// TIA Portal V19 export
FUNCTION "RO_2" : Void   // FC11, LAD
{ S7_Optimized_Access := 'TRUE' }
// stored: SetENOAutomatically false
   VAR_TEMP   // added for the SCL form of the ladder/FBD networks
      _w1 : Bool;
   END_VAR
BEGIN

REGION Network 1: FEED PUMP
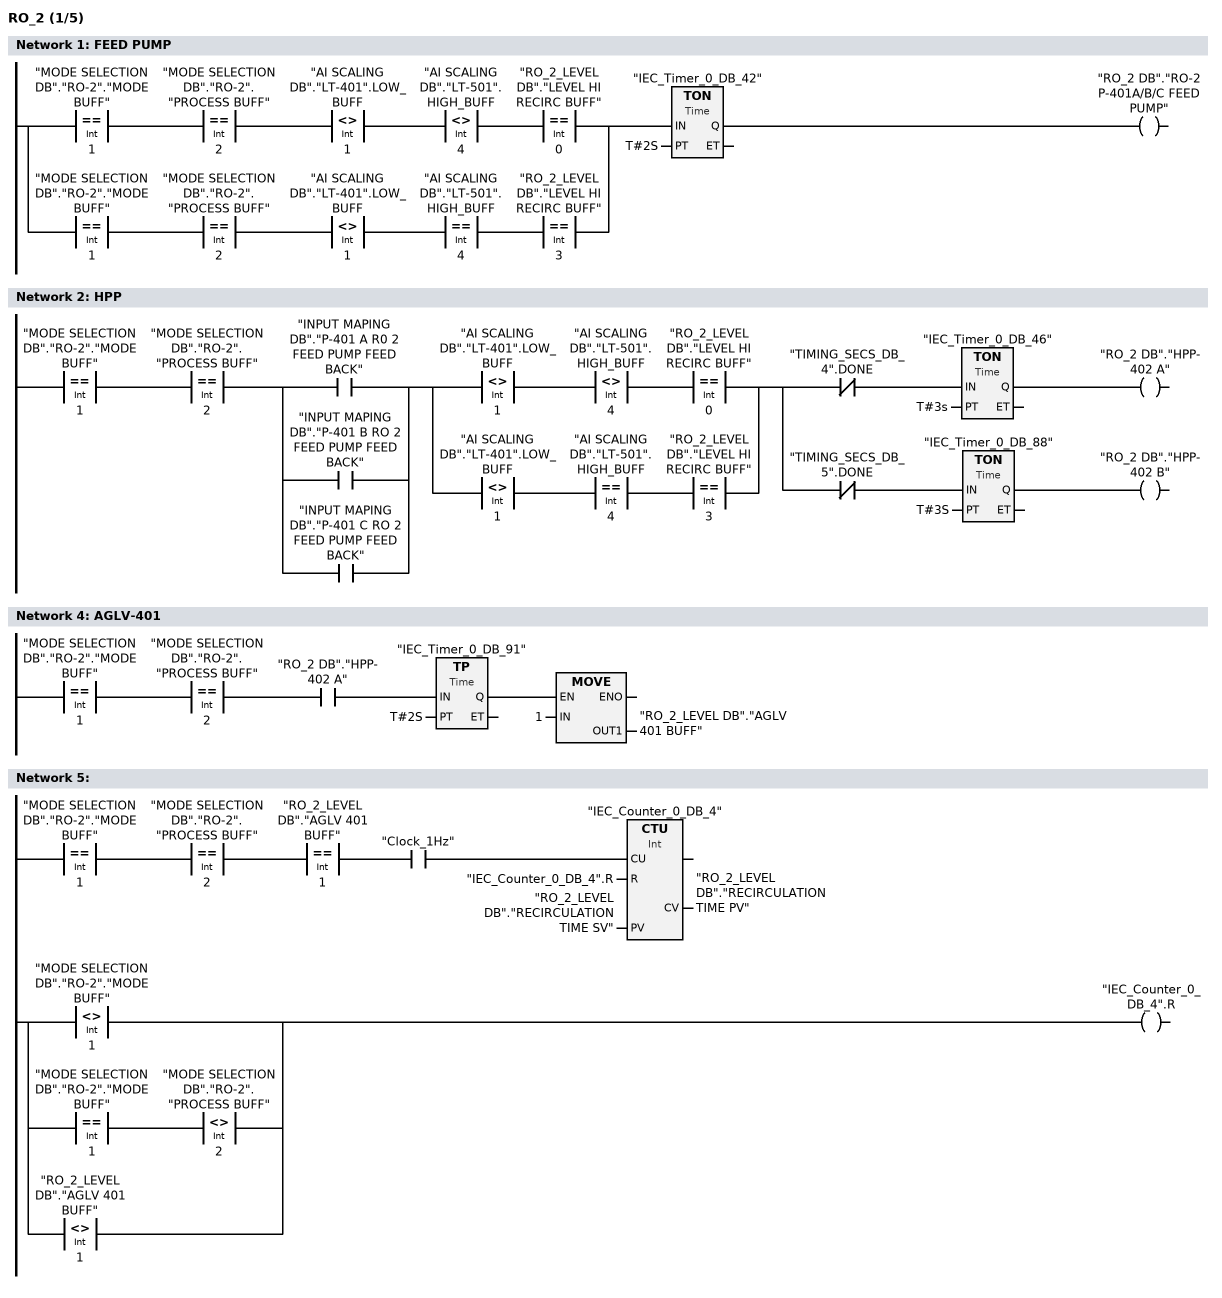
   RUNG wire#powerrail
      { S7_Templates := "SrcType := Int" } EQ_Contact(in1 := "MODE SELECTION DB"."RO-2"."MODE BUFF", in2 := 1)
      { S7_Templates := "SrcType := Int" } EQ_Contact(in1 := "MODE SELECTION DB"."RO-2"."PROCESS BUFF", in2 := 2)
      { S7_Templates := "SrcType := Int" } NE_Contact(in1 := "AI SCALING DB"."LT-401".LOW_BUFF, in2 := 1)
      { S7_Templates := "SrcType := Int" } NE_Contact(in1 := "AI SCALING DB"."LT-501".HIGH_BUFF, in2 := 4)
      { S7_Templates := "SrcType := Int" } EQ_Contact(in1 := "RO_2_LEVEL DB"."LEVEL HI RECIRC BUFF", in2 := 0)
      wire#w1
      { S7_Templates := "time_type := Time" } "IEC_Timer_0_DB_42".TON(pt := T#2S, et =>)
      Coil( "RO_2 DB"."RO-2 P-401A/B/C FEED PUMP" )
   END_RUNG
   RUNG wire#powerrail
      { S7_Templates := "SrcType := Int" } EQ_Contact(in1 := "MODE SELECTION DB"."RO-2"."MODE BUFF", in2 := 1)
      { S7_Templates := "SrcType := Int" } EQ_Contact(in1 := "MODE SELECTION DB"."RO-2"."PROCESS BUFF", in2 := 2)
      { S7_Templates := "SrcType := Int" } NE_Contact(in1 := "AI SCALING DB"."LT-401".LOW_BUFF, in2 := 1)
      { S7_Templates := "SrcType := Int" } EQ_Contact(in1 := "AI SCALING DB"."LT-501".HIGH_BUFF, in2 := 4)
      { S7_Templates := "SrcType := Int" } EQ_Contact(in1 := "RO_2_LEVEL DB"."LEVEL HI RECIRC BUFF", in2 := 3)
   END_RUNG wire#w1
   // the same network as SCL:
   "IEC_Timer_0_DB_42".TON(IN := (("MODE SELECTION DB"."RO-2"."MODE BUFF" = 1) AND ("MODE SELECTION DB"."RO-2"."PROCESS BUFF" = 2) AND ("AI SCALING DB"."LT-401".LOW_BUFF <> 1) AND ("AI SCALING DB"."LT-501".HIGH_BUFF <> 4) AND ("RO_2_LEVEL DB"."LEVEL HI RECIRC BUFF" = 0)) OR (("MODE SELECTION DB"."RO-2"."MODE BUFF" = 1) AND ("MODE SELECTION DB"."RO-2"."PROCESS BUFF" = 2) AND ("AI SCALING DB"."LT-401".LOW_BUFF <> 1) AND ("AI SCALING DB"."LT-501".HIGH_BUFF = 4) AND ("RO_2_LEVEL DB"."LEVEL HI RECIRC BUFF" = 3)),
                           PT := T#2S);
   "RO_2 DB"."RO-2 P-401A/B/C FEED PUMP" := "IEC_Timer_0_DB_42".Q;
END_REGION

REGION Network 2: HPP
   RUNG wire#powerrail
      { S7_Templates := "SrcType := Int" } EQ_Contact(in1 := "MODE SELECTION DB"."RO-2"."MODE BUFF", in2 := 1)
      { S7_Templates := "SrcType := Int" } EQ_Contact(in1 := "MODE SELECTION DB"."RO-2"."PROCESS BUFF", in2 := 2)
      wire#w1
      Contact( "INPUT MAPING DB"."P-401 A R0 2 FEED PUMP FEED BACK" )
      wire#w2
      { S7_Templates := "SrcType := Int" } NE_Contact(in1 := "AI SCALING DB"."LT-401".LOW_BUFF, in2 := 1)
      { S7_Templates := "SrcType := Int" } NE_Contact(in1 := "AI SCALING DB"."LT-501".HIGH_BUFF, in2 := 4)
      { S7_Templates := "SrcType := Int" } EQ_Contact(in1 := "RO_2_LEVEL DB"."LEVEL HI RECIRC BUFF", in2 := 0)
      wire#w3
      I_Contact( "TIMING_SECS_DB_4".DONE )
      { S7_Templates := "time_type := Time" } "IEC_Timer_0_DB_46".TON(pt := T#3s, et =>)
      Coil( "RO_2 DB"."HPP-402 A" )
   END_RUNG
   RUNG wire#w1
      Contact( "INPUT MAPING DB"."P-401 B RO 2 FEED PUMP FEED BACK" )
   END_RUNG wire#w2
   RUNG wire#w1
      Contact( "INPUT MAPING DB"."P-401 C RO 2 FEED PUMP FEED BACK" )
   END_RUNG wire#w2
   RUNG wire#w2
      { S7_Templates := "SrcType := Int" } NE_Contact(in1 := "AI SCALING DB"."LT-401".LOW_BUFF, in2 := 1)
      { S7_Templates := "SrcType := Int" } EQ_Contact(in1 := "AI SCALING DB"."LT-501".HIGH_BUFF, in2 := 4)
      { S7_Templates := "SrcType := Int" } EQ_Contact(in1 := "RO_2_LEVEL DB"."LEVEL HI RECIRC BUFF", in2 := 3)
   END_RUNG wire#w3
   RUNG wire#w3
      I_Contact( "TIMING_SECS_DB_5".DONE )
      { S7_Templates := "time_type := Time" } "IEC_Timer_0_DB_88".TON(pt := T#3S, et =>)
      Coil( "RO_2 DB"."HPP-402 B" )
   END_RUNG
   // the same network as SCL:
   #_w1 := ("MODE SELECTION DB"."RO-2"."MODE BUFF" = 1) AND ("MODE SELECTION DB"."RO-2"."PROCESS BUFF" = 2) AND ("INPUT MAPING DB"."P-401 A R0 2 FEED PUMP FEED BACK" OR "INPUT MAPING DB"."P-401 B RO 2 FEED PUMP FEED BACK" OR "INPUT MAPING DB"."P-401 C RO 2 FEED PUMP FEED BACK") AND ((("AI SCALING DB"."LT-401".LOW_BUFF <> 1) AND ("AI SCALING DB"."LT-501".HIGH_BUFF <> 4) AND ("RO_2_LEVEL DB"."LEVEL HI RECIRC BUFF" = 0)) OR (("AI SCALING DB"."LT-401".LOW_BUFF <> 1) AND ("AI SCALING DB"."LT-501".HIGH_BUFF = 4) AND ("RO_2_LEVEL DB"."LEVEL HI RECIRC BUFF" = 3)));
   "IEC_Timer_0_DB_46".TON(IN := #_w1 AND NOT "TIMING_SECS_DB_4".DONE, PT := T#3s);
   "RO_2 DB"."HPP-402 A" := "IEC_Timer_0_DB_46".Q;
   "IEC_Timer_0_DB_88".TON(IN := #_w1 AND NOT "TIMING_SECS_DB_5".DONE, PT := T#3S);
   "RO_2 DB"."HPP-402 B" := "IEC_Timer_0_DB_88".Q;
END_REGION

REGION Network 4: AGLV-401
   RUNG wire#powerrail
      { S7_Templates := "SrcType := Int" } EQ_Contact(in1 := "MODE SELECTION DB"."RO-2"."MODE BUFF", in2 := 1)
      { S7_Templates := "SrcType := Int" } EQ_Contact(in1 := "MODE SELECTION DB"."RO-2"."PROCESS BUFF", in2 := 2)
      Contact( "RO_2 DB"."HPP-402 A" )
      { S7_Templates := "time_type := Time" } "IEC_Timer_0_DB_91".TP(pt := T#2S, et =>)
      Move(in := 1, out1 => "RO_2_LEVEL DB"."AGLV 401 BUFF")
   END_RUNG
   // the same network as SCL:
   "IEC_Timer_0_DB_91".TP(IN := ("MODE SELECTION DB"."RO-2"."MODE BUFF" = 1) AND ("MODE SELECTION DB"."RO-2"."PROCESS BUFF" = 2) AND "RO_2 DB"."HPP-402 A",
                          PT := T#2S);
   IF "IEC_Timer_0_DB_91".Q THEN "RO_2_LEVEL DB"."AGLV 401 BUFF" := 1; END_IF;
END_REGION

REGION Network 5
   RUNG wire#powerrail
      { S7_Templates := "SrcType := Int" } EQ_Contact(in1 := "MODE SELECTION DB"."RO-2"."MODE BUFF", in2 := 1)
      { S7_Templates := "SrcType := Int" } EQ_Contact(in1 := "MODE SELECTION DB"."RO-2"."PROCESS BUFF", in2 := 2)
      { S7_Templates := "SrcType := Int" } EQ_Contact(in1 := "RO_2_LEVEL DB"."AGLV 401 BUFF", in2 := 1)
      Contact( "Clock_1Hz" )
      { S7_Templates := "value_type := Int" } "IEC_Counter_0_DB_4".CTU(r := "IEC_Counter_0_DB_4".R, pv := "RO_2_LEVEL DB"."RECIRCULATION TIME SV", cv => "RO_2_LEVEL DB"."RECIRCULATION TIME PV")
   END_RUNG
   RUNG wire#powerrail
      { S7_Templates := "SrcType := Int" } NE_Contact(in1 := "MODE SELECTION DB"."RO-2"."MODE BUFF", in2 := 1)
      wire#w1
      Coil( "IEC_Counter_0_DB_4".R )
   END_RUNG
   RUNG wire#powerrail
      { S7_Templates := "SrcType := Int" } EQ_Contact(in1 := "MODE SELECTION DB"."RO-2"."MODE BUFF", in2 := 1)
      { S7_Templates := "SrcType := Int" } NE_Contact(in1 := "MODE SELECTION DB"."RO-2"."PROCESS BUFF", in2 := 2)
   END_RUNG wire#w1
   RUNG wire#powerrail
      { S7_Templates := "SrcType := Int" } NE_Contact(in1 := "RO_2_LEVEL DB"."AGLV 401 BUFF", in2 := 1)
   END_RUNG wire#w1
   // the same network as SCL:
   "IEC_Counter_0_DB_4".CTU(CU := ("MODE SELECTION DB"."RO-2"."MODE BUFF" = 1) AND ("MODE SELECTION DB"."RO-2"."PROCESS BUFF" = 2) AND ("RO_2_LEVEL DB"."AGLV 401 BUFF" = 1) AND "Clock_1Hz",
                           R := "IEC_Counter_0_DB_4".R,
                           PV := "RO_2_LEVEL DB"."RECIRCULATION TIME SV",
                           CV => "RO_2_LEVEL DB"."RECIRCULATION TIME PV");
   "IEC_Counter_0_DB_4".R := ("MODE SELECTION DB"."RO-2"."MODE BUFF" <> 1) OR (("MODE SELECTION DB"."RO-2"."MODE BUFF" = 1) AND ("MODE SELECTION DB"."RO-2"."PROCESS BUFF" <> 2)) OR ("RO_2_LEVEL DB"."AGLV 401 BUFF" <> 1);
END_REGION

REGION Network 6
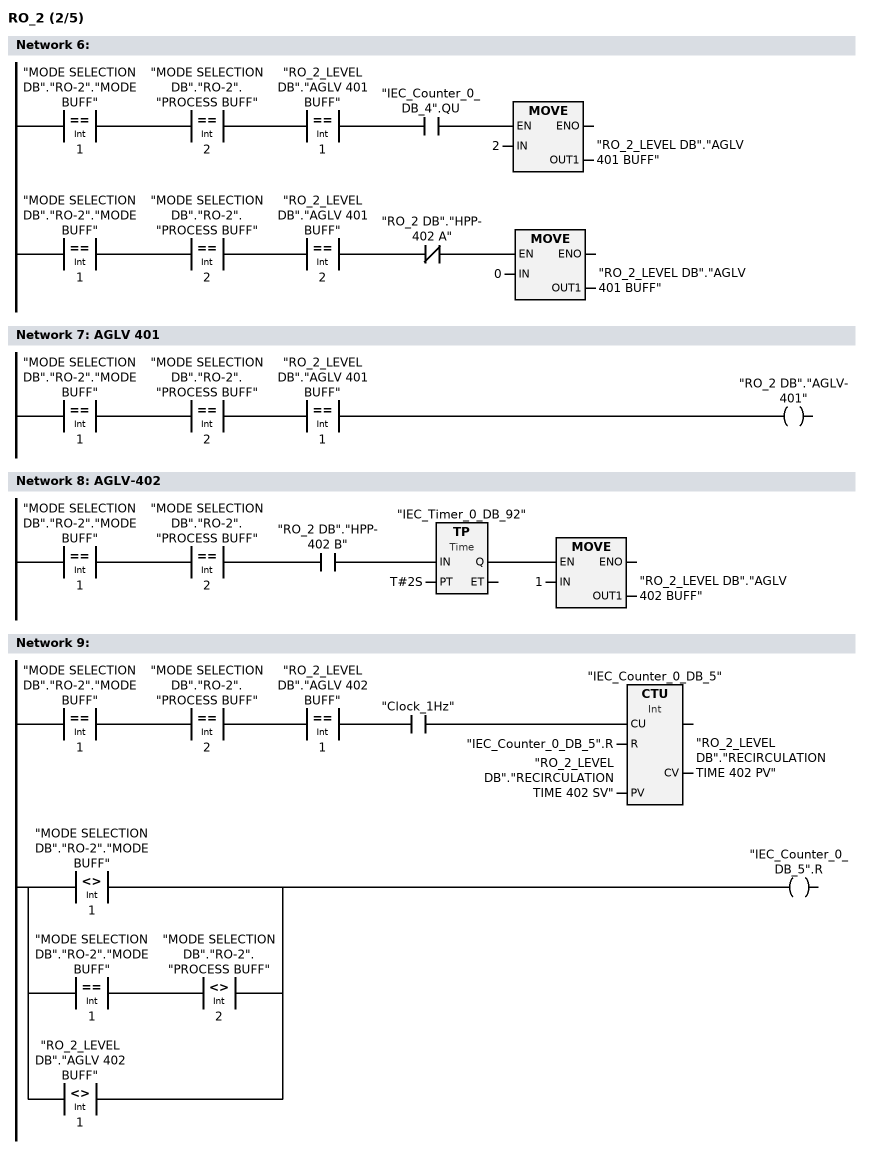
   RUNG wire#powerrail
      { S7_Templates := "SrcType := Int" } EQ_Contact(in1 := "MODE SELECTION DB"."RO-2"."MODE BUFF", in2 := 1)
      { S7_Templates := "SrcType := Int" } EQ_Contact(in1 := "MODE SELECTION DB"."RO-2"."PROCESS BUFF", in2 := 2)
      { S7_Templates := "SrcType := Int" } EQ_Contact(in1 := "RO_2_LEVEL DB"."AGLV 401 BUFF", in2 := 1)
      Contact( "IEC_Counter_0_DB_4".QU )
      Move(in := 2, out1 => "RO_2_LEVEL DB"."AGLV 401 BUFF")
   END_RUNG
   RUNG wire#powerrail
      { S7_Templates := "SrcType := Int" } EQ_Contact(in1 := "MODE SELECTION DB"."RO-2"."MODE BUFF", in2 := 1)
      { S7_Templates := "SrcType := Int" } EQ_Contact(in1 := "MODE SELECTION DB"."RO-2"."PROCESS BUFF", in2 := 2)
      { S7_Templates := "SrcType := Int" } EQ_Contact(in1 := "RO_2_LEVEL DB"."AGLV 401 BUFF", in2 := 2)
      I_Contact( "RO_2 DB"."HPP-402 A" )
      Move(in := 0, out1 => "RO_2_LEVEL DB"."AGLV 401 BUFF")
   END_RUNG
   // the same network as SCL:
   IF ("MODE SELECTION DB"."RO-2"."MODE BUFF" = 1) AND ("MODE SELECTION DB"."RO-2"."PROCESS BUFF" = 2) AND ("RO_2_LEVEL DB"."AGLV 401 BUFF" = 1) AND "IEC_Counter_0_DB_4".QU THEN
       "RO_2_LEVEL DB"."AGLV 401 BUFF" := 2;
   END_IF;
   IF ("MODE SELECTION DB"."RO-2"."MODE BUFF" = 1) AND ("MODE SELECTION DB"."RO-2"."PROCESS BUFF" = 2) AND ("RO_2_LEVEL DB"."AGLV 401 BUFF" = 2) AND NOT "RO_2 DB"."HPP-402 A" THEN
       "RO_2_LEVEL DB"."AGLV 401 BUFF" := 0;
   END_IF;
END_REGION

REGION Network 7: AGLV 401
   RUNG wire#powerrail
      { S7_Templates := "SrcType := Int" } EQ_Contact(in1 := "MODE SELECTION DB"."RO-2"."MODE BUFF", in2 := 1)
      { S7_Templates := "SrcType := Int" } EQ_Contact(in1 := "MODE SELECTION DB"."RO-2"."PROCESS BUFF", in2 := 2)
      { S7_Templates := "SrcType := Int" } EQ_Contact(in1 := "RO_2_LEVEL DB"."AGLV 401 BUFF", in2 := 1)
      Coil( "RO_2 DB"."AGLV-401" )
   END_RUNG
   // the same network as SCL:
   "RO_2 DB"."AGLV-401" := ("MODE SELECTION DB"."RO-2"."MODE BUFF" = 1) AND ("MODE SELECTION DB"."RO-2"."PROCESS BUFF" = 2) AND ("RO_2_LEVEL DB"."AGLV 401 BUFF" = 1);
END_REGION

REGION Network 8: AGLV-402
   RUNG wire#powerrail
      { S7_Templates := "SrcType := Int" } EQ_Contact(in1 := "MODE SELECTION DB"."RO-2"."MODE BUFF", in2 := 1)
      { S7_Templates := "SrcType := Int" } EQ_Contact(in1 := "MODE SELECTION DB"."RO-2"."PROCESS BUFF", in2 := 2)
      Contact( "RO_2 DB"."HPP-402 B" )
      { S7_Templates := "time_type := Time" } "IEC_Timer_0_DB_92".TP(pt := T#2S, et =>)
      Move(in := 1, out1 => "RO_2_LEVEL DB"."AGLV 402 BUFF")
   END_RUNG
   // the same network as SCL:
   "IEC_Timer_0_DB_92".TP(IN := ("MODE SELECTION DB"."RO-2"."MODE BUFF" = 1) AND ("MODE SELECTION DB"."RO-2"."PROCESS BUFF" = 2) AND "RO_2 DB"."HPP-402 B",
                          PT := T#2S);
   IF "IEC_Timer_0_DB_92".Q THEN "RO_2_LEVEL DB"."AGLV 402 BUFF" := 1; END_IF;
END_REGION

REGION Network 9
   RUNG wire#powerrail
      { S7_Templates := "SrcType := Int" } EQ_Contact(in1 := "MODE SELECTION DB"."RO-2"."MODE BUFF", in2 := 1)
      { S7_Templates := "SrcType := Int" } EQ_Contact(in1 := "MODE SELECTION DB"."RO-2"."PROCESS BUFF", in2 := 2)
      { S7_Templates := "SrcType := Int" } EQ_Contact(in1 := "RO_2_LEVEL DB"."AGLV 402 BUFF", in2 := 1)
      Contact( "Clock_1Hz" )
      { S7_Templates := "value_type := Int" } "IEC_Counter_0_DB_5".CTU(r := "IEC_Counter_0_DB_5".R, pv := "RO_2_LEVEL DB"."RECIRCULATION TIME 402 SV", cv => "RO_2_LEVEL DB"."RECIRCULATION TIME 402 PV")
   END_RUNG
   RUNG wire#powerrail
      { S7_Templates := "SrcType := Int" } NE_Contact(in1 := "MODE SELECTION DB"."RO-2"."MODE BUFF", in2 := 1)
      wire#w1
      Coil( "IEC_Counter_0_DB_5".R )
   END_RUNG
   RUNG wire#powerrail
      { S7_Templates := "SrcType := Int" } EQ_Contact(in1 := "MODE SELECTION DB"."RO-2"."MODE BUFF", in2 := 1)
      { S7_Templates := "SrcType := Int" } NE_Contact(in1 := "MODE SELECTION DB"."RO-2"."PROCESS BUFF", in2 := 2)
   END_RUNG wire#w1
   RUNG wire#powerrail
      { S7_Templates := "SrcType := Int" } NE_Contact(in1 := "RO_2_LEVEL DB"."AGLV 402 BUFF", in2 := 1)
   END_RUNG wire#w1
   // the same network as SCL:
   "IEC_Counter_0_DB_5".CTU(CU := ("MODE SELECTION DB"."RO-2"."MODE BUFF" = 1) AND ("MODE SELECTION DB"."RO-2"."PROCESS BUFF" = 2) AND ("RO_2_LEVEL DB"."AGLV 402 BUFF" = 1) AND "Clock_1Hz",
                           R := "IEC_Counter_0_DB_5".R,
                           PV := "RO_2_LEVEL DB"."RECIRCULATION TIME 402 SV",
                           CV => "RO_2_LEVEL DB"."RECIRCULATION TIME 402 PV");
   "IEC_Counter_0_DB_5".R := ("MODE SELECTION DB"."RO-2"."MODE BUFF" <> 1) OR (("MODE SELECTION DB"."RO-2"."MODE BUFF" = 1) AND ("MODE SELECTION DB"."RO-2"."PROCESS BUFF" <> 2)) OR ("RO_2_LEVEL DB"."AGLV 402 BUFF" <> 1);
END_REGION

REGION Network 10
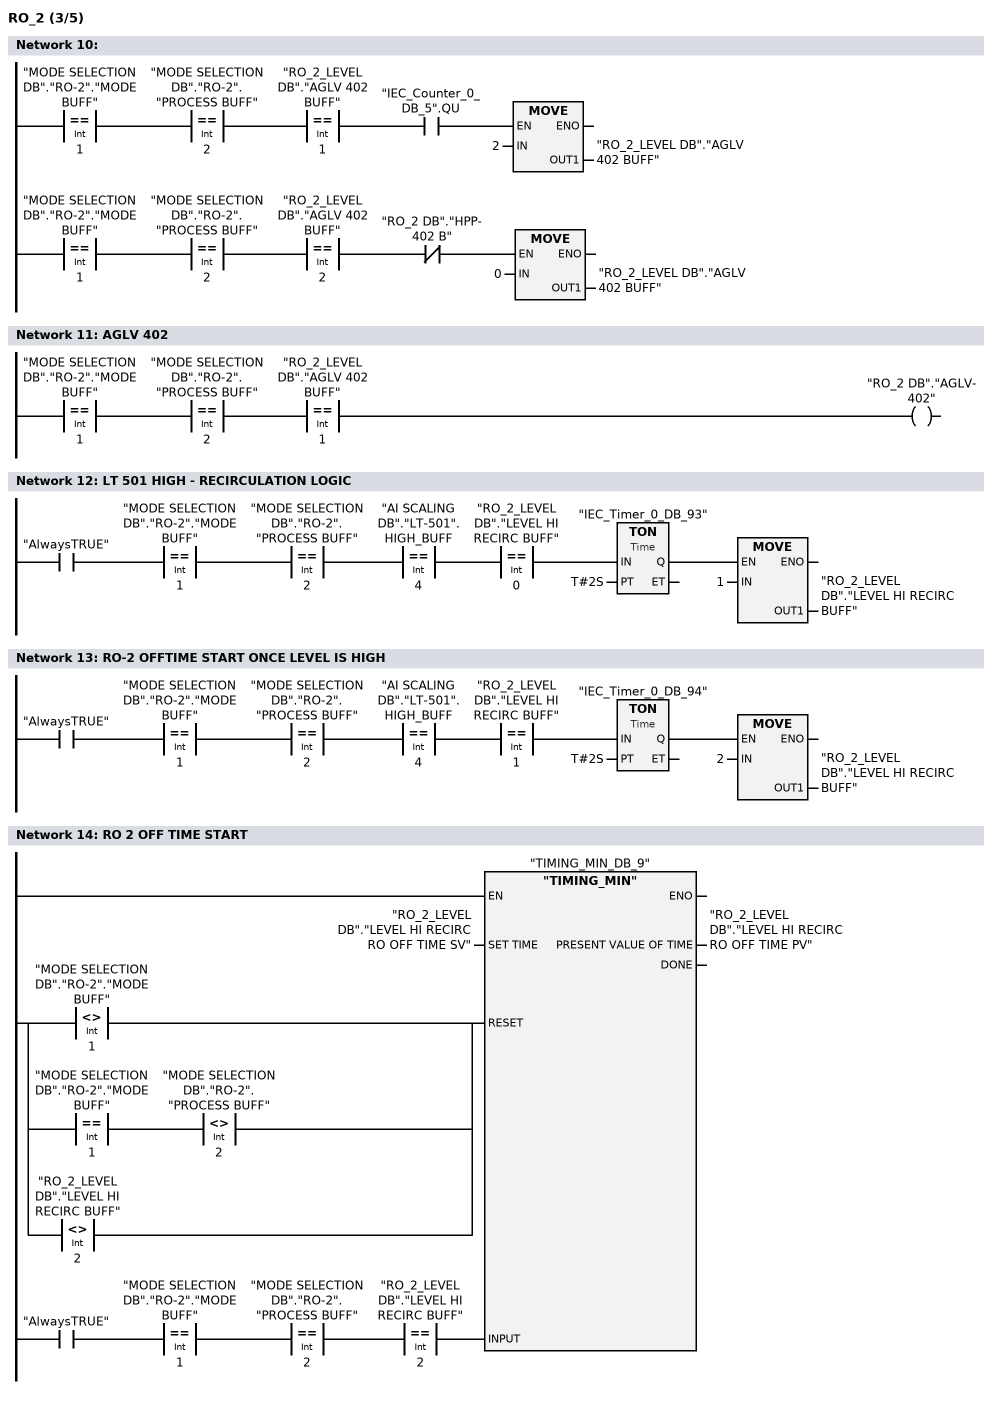
   RUNG wire#powerrail
      { S7_Templates := "SrcType := Int" } EQ_Contact(in1 := "MODE SELECTION DB"."RO-2"."MODE BUFF", in2 := 1)
      { S7_Templates := "SrcType := Int" } EQ_Contact(in1 := "MODE SELECTION DB"."RO-2"."PROCESS BUFF", in2 := 2)
      { S7_Templates := "SrcType := Int" } EQ_Contact(in1 := "RO_2_LEVEL DB"."AGLV 402 BUFF", in2 := 1)
      Contact( "IEC_Counter_0_DB_5".QU )
      Move(in := 2, out1 => "RO_2_LEVEL DB"."AGLV 402 BUFF")
   END_RUNG
   RUNG wire#powerrail
      { S7_Templates := "SrcType := Int" } EQ_Contact(in1 := "MODE SELECTION DB"."RO-2"."MODE BUFF", in2 := 1)
      { S7_Templates := "SrcType := Int" } EQ_Contact(in1 := "MODE SELECTION DB"."RO-2"."PROCESS BUFF", in2 := 2)
      { S7_Templates := "SrcType := Int" } EQ_Contact(in1 := "RO_2_LEVEL DB"."AGLV 402 BUFF", in2 := 2)
      I_Contact( "RO_2 DB"."HPP-402 B" )
      Move(in := 0, out1 => "RO_2_LEVEL DB"."AGLV 402 BUFF")
   END_RUNG
   // the same network as SCL:
   IF ("MODE SELECTION DB"."RO-2"."MODE BUFF" = 1) AND ("MODE SELECTION DB"."RO-2"."PROCESS BUFF" = 2) AND ("RO_2_LEVEL DB"."AGLV 402 BUFF" = 1) AND "IEC_Counter_0_DB_5".QU THEN
       "RO_2_LEVEL DB"."AGLV 402 BUFF" := 2;
   END_IF;
   IF ("MODE SELECTION DB"."RO-2"."MODE BUFF" = 1) AND ("MODE SELECTION DB"."RO-2"."PROCESS BUFF" = 2) AND ("RO_2_LEVEL DB"."AGLV 402 BUFF" = 2) AND NOT "RO_2 DB"."HPP-402 B" THEN
       "RO_2_LEVEL DB"."AGLV 402 BUFF" := 0;
   END_IF;
END_REGION

REGION Network 11: AGLV 402
   RUNG wire#powerrail
      { S7_Templates := "SrcType := Int" } EQ_Contact(in1 := "MODE SELECTION DB"."RO-2"."MODE BUFF", in2 := 1)
      { S7_Templates := "SrcType := Int" } EQ_Contact(in1 := "MODE SELECTION DB"."RO-2"."PROCESS BUFF", in2 := 2)
      { S7_Templates := "SrcType := Int" } EQ_Contact(in1 := "RO_2_LEVEL DB"."AGLV 402 BUFF", in2 := 1)
      Coil( "RO_2 DB"."AGLV-402" )
   END_RUNG
   // the same network as SCL:
   "RO_2 DB"."AGLV-402" := ("MODE SELECTION DB"."RO-2"."MODE BUFF" = 1) AND ("MODE SELECTION DB"."RO-2"."PROCESS BUFF" = 2) AND ("RO_2_LEVEL DB"."AGLV 402 BUFF" = 1);
END_REGION

REGION Network 12: LT 501 HIGH - RECIRCULATION LOGIC
   RUNG wire#powerrail
      Contact( "AlwaysTRUE" )
      { S7_Templates := "SrcType := Int" } EQ_Contact(in1 := "MODE SELECTION DB"."RO-2"."MODE BUFF", in2 := 1)
      { S7_Templates := "SrcType := Int" } EQ_Contact(in1 := "MODE SELECTION DB"."RO-2"."PROCESS BUFF", in2 := 2)
      { S7_Templates := "SrcType := Int" } EQ_Contact(in1 := "AI SCALING DB"."LT-501".HIGH_BUFF, in2 := 4)
      { S7_Templates := "SrcType := Int" } EQ_Contact(in1 := "RO_2_LEVEL DB"."LEVEL HI RECIRC BUFF", in2 := 0)
      { S7_Templates := "time_type := Time" } "IEC_Timer_0_DB_93".TON(pt := T#2S, et =>)
      Move(in := 1, out1 => "RO_2_LEVEL DB"."LEVEL HI RECIRC BUFF")
   END_RUNG
   // the same network as SCL:
   "IEC_Timer_0_DB_93".TON(IN := "AlwaysTRUE" AND ("MODE SELECTION DB"."RO-2"."MODE BUFF" = 1) AND ("MODE SELECTION DB"."RO-2"."PROCESS BUFF" = 2) AND ("AI SCALING DB"."LT-501".HIGH_BUFF = 4) AND ("RO_2_LEVEL DB"."LEVEL HI RECIRC BUFF" = 0),
                           PT := T#2S);
   IF "IEC_Timer_0_DB_93".Q THEN "RO_2_LEVEL DB"."LEVEL HI RECIRC BUFF" := 1; END_IF;
END_REGION

REGION Network 13: RO-2 OFFTIME START ONCE LEVEL IS HIGH
   RUNG wire#powerrail
      Contact( "AlwaysTRUE" )
      { S7_Templates := "SrcType := Int" } EQ_Contact(in1 := "MODE SELECTION DB"."RO-2"."MODE BUFF", in2 := 1)
      { S7_Templates := "SrcType := Int" } EQ_Contact(in1 := "MODE SELECTION DB"."RO-2"."PROCESS BUFF", in2 := 2)
      { S7_Templates := "SrcType := Int" } EQ_Contact(in1 := "AI SCALING DB"."LT-501".HIGH_BUFF, in2 := 4)
      { S7_Templates := "SrcType := Int" } EQ_Contact(in1 := "RO_2_LEVEL DB"."LEVEL HI RECIRC BUFF", in2 := 1)
      { S7_Templates := "time_type := Time" } "IEC_Timer_0_DB_94".TON(pt := T#2S, et =>)
      Move(in := 2, out1 => "RO_2_LEVEL DB"."LEVEL HI RECIRC BUFF")
   END_RUNG
   // the same network as SCL:
   "IEC_Timer_0_DB_94".TON(IN := "AlwaysTRUE" AND ("MODE SELECTION DB"."RO-2"."MODE BUFF" = 1) AND ("MODE SELECTION DB"."RO-2"."PROCESS BUFF" = 2) AND ("AI SCALING DB"."LT-501".HIGH_BUFF = 4) AND ("RO_2_LEVEL DB"."LEVEL HI RECIRC BUFF" = 1),
                           PT := T#2S);
   IF "IEC_Timer_0_DB_94".Q THEN "RO_2_LEVEL DB"."LEVEL HI RECIRC BUFF" := 2; END_IF;
END_REGION

REGION Network 14: RO 2 OFF TIME START
   RUNG wire#powerrail
      "TIMING_MIN_DB_9"(RESET := wire#w1, INPUT := wire#w2, "SET TIME" := "RO_2_LEVEL DB"."LEVEL HI RECIRC RO OFF TIME SV", "PRESENT VALUE OF TIME" => "RO_2_LEVEL DB"."LEVEL HI RECIRC RO OFF TIME PV", DONE =>)
   END_RUNG
   RUNG wire#powerrail
      { S7_Templates := "SrcType := Int" } NE_Contact(in1 := "MODE SELECTION DB"."RO-2"."MODE BUFF", in2 := 1)
   END_RUNG wire#w1
   RUNG wire#powerrail
      { S7_Templates := "SrcType := Int" } EQ_Contact(in1 := "MODE SELECTION DB"."RO-2"."MODE BUFF", in2 := 1)
      { S7_Templates := "SrcType := Int" } NE_Contact(in1 := "MODE SELECTION DB"."RO-2"."PROCESS BUFF", in2 := 2)
   END_RUNG wire#w1
   RUNG wire#powerrail
      { S7_Templates := "SrcType := Int" } NE_Contact(in1 := "RO_2_LEVEL DB"."LEVEL HI RECIRC BUFF", in2 := 2)
   END_RUNG wire#w1
   RUNG wire#powerrail
      Contact( "AlwaysTRUE" )
      { S7_Templates := "SrcType := Int" } EQ_Contact(in1 := "MODE SELECTION DB"."RO-2"."MODE BUFF", in2 := 1)
      { S7_Templates := "SrcType := Int" } EQ_Contact(in1 := "MODE SELECTION DB"."RO-2"."PROCESS BUFF", in2 := 2)
      { S7_Templates := "SrcType := Int" } EQ_Contact(in1 := "RO_2_LEVEL DB"."LEVEL HI RECIRC BUFF", in2 := 2)
   END_RUNG wire#w2
   // the same network as SCL:
   "TIMING_MIN_DB_9"("SET TIME" := "RO_2_LEVEL DB"."LEVEL HI RECIRC RO OFF TIME SV",   // "TIMING_MIN"
                     RESET := ("MODE SELECTION DB"."RO-2"."MODE BUFF" <> 1) OR (("MODE SELECTION DB"."RO-2"."MODE BUFF" = 1) AND ("MODE SELECTION DB"."RO-2"."PROCESS BUFF" <> 2)) OR ("RO_2_LEVEL DB"."LEVEL HI RECIRC BUFF" <> 2),
                     INPUT := "AlwaysTRUE" AND ("MODE SELECTION DB"."RO-2"."MODE BUFF" = 1) AND ("MODE SELECTION DB"."RO-2"."PROCESS BUFF" = 2) AND ("RO_2_LEVEL DB"."LEVEL HI RECIRC BUFF" = 2),
                     "PRESENT VALUE OF TIME" => "RO_2_LEVEL DB"."LEVEL HI RECIRC RO OFF TIME PV");
END_REGION

REGION Network 15: RO 2 RECIRCULATION START AFTER OFF TIME OVER
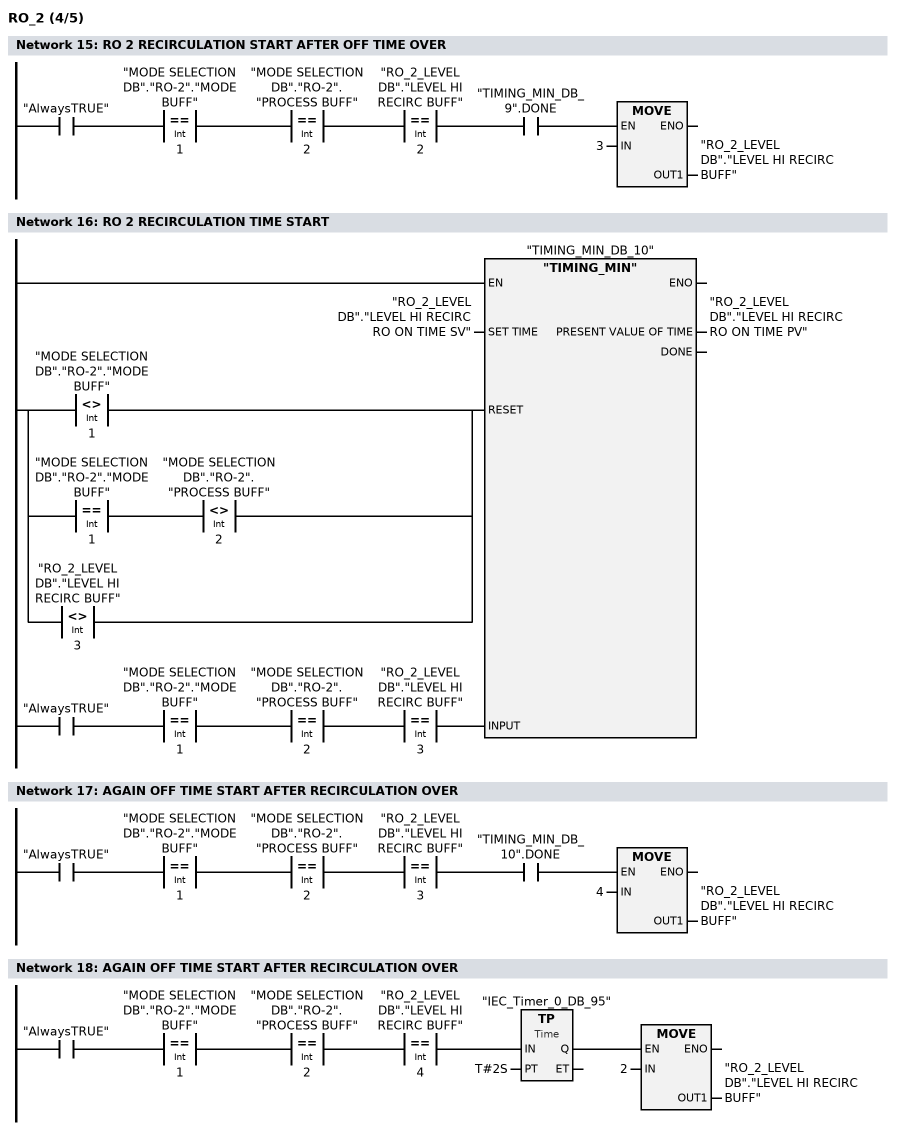
   RUNG wire#powerrail
      Contact( "AlwaysTRUE" )
      { S7_Templates := "SrcType := Int" } EQ_Contact(in1 := "MODE SELECTION DB"."RO-2"."MODE BUFF", in2 := 1)
      { S7_Templates := "SrcType := Int" } EQ_Contact(in1 := "MODE SELECTION DB"."RO-2"."PROCESS BUFF", in2 := 2)
      { S7_Templates := "SrcType := Int" } EQ_Contact(in1 := "RO_2_LEVEL DB"."LEVEL HI RECIRC BUFF", in2 := 2)
      Contact( "TIMING_MIN_DB_9".DONE )
      Move(in := 3, out1 => "RO_2_LEVEL DB"."LEVEL HI RECIRC BUFF")
   END_RUNG
   // the same network as SCL:
   IF "AlwaysTRUE" AND ("MODE SELECTION DB"."RO-2"."MODE BUFF" = 1) AND ("MODE SELECTION DB"."RO-2"."PROCESS BUFF" = 2) AND ("RO_2_LEVEL DB"."LEVEL HI RECIRC BUFF" = 2) AND "TIMING_MIN_DB_9".DONE THEN
       "RO_2_LEVEL DB"."LEVEL HI RECIRC BUFF" := 3;
   END_IF;
END_REGION

REGION Network 16: RO 2 RECIRCULATION TIME START
   RUNG wire#powerrail
      "TIMING_MIN_DB_10"(RESET := wire#w1, INPUT := wire#w2, "SET TIME" := "RO_2_LEVEL DB"."LEVEL HI RECIRC RO ON TIME SV", "PRESENT VALUE OF TIME" => "RO_2_LEVEL DB"."LEVEL HI RECIRC RO ON TIME PV", DONE =>)
   END_RUNG
   RUNG wire#powerrail
      { S7_Templates := "SrcType := Int" } NE_Contact(in1 := "MODE SELECTION DB"."RO-2"."MODE BUFF", in2 := 1)
   END_RUNG wire#w1
   RUNG wire#powerrail
      { S7_Templates := "SrcType := Int" } EQ_Contact(in1 := "MODE SELECTION DB"."RO-2"."MODE BUFF", in2 := 1)
      { S7_Templates := "SrcType := Int" } NE_Contact(in1 := "MODE SELECTION DB"."RO-2"."PROCESS BUFF", in2 := 2)
   END_RUNG wire#w1
   RUNG wire#powerrail
      { S7_Templates := "SrcType := Int" } NE_Contact(in1 := "RO_2_LEVEL DB"."LEVEL HI RECIRC BUFF", in2 := 3)
   END_RUNG wire#w1
   RUNG wire#powerrail
      Contact( "AlwaysTRUE" )
      { S7_Templates := "SrcType := Int" } EQ_Contact(in1 := "MODE SELECTION DB"."RO-2"."MODE BUFF", in2 := 1)
      { S7_Templates := "SrcType := Int" } EQ_Contact(in1 := "MODE SELECTION DB"."RO-2"."PROCESS BUFF", in2 := 2)
      { S7_Templates := "SrcType := Int" } EQ_Contact(in1 := "RO_2_LEVEL DB"."LEVEL HI RECIRC BUFF", in2 := 3)
   END_RUNG wire#w2
   // the same network as SCL:
   "TIMING_MIN_DB_10"("SET TIME" := "RO_2_LEVEL DB"."LEVEL HI RECIRC RO ON TIME SV",   // "TIMING_MIN"
                      RESET := ("MODE SELECTION DB"."RO-2"."MODE BUFF" <> 1) OR (("MODE SELECTION DB"."RO-2"."MODE BUFF" = 1) AND ("MODE SELECTION DB"."RO-2"."PROCESS BUFF" <> 2)) OR ("RO_2_LEVEL DB"."LEVEL HI RECIRC BUFF" <> 3),
                      INPUT := "AlwaysTRUE" AND ("MODE SELECTION DB"."RO-2"."MODE BUFF" = 1) AND ("MODE SELECTION DB"."RO-2"."PROCESS BUFF" = 2) AND ("RO_2_LEVEL DB"."LEVEL HI RECIRC BUFF" = 3),
                      "PRESENT VALUE OF TIME" => "RO_2_LEVEL DB"."LEVEL HI RECIRC RO ON TIME PV");
END_REGION

REGION Network 17: AGAIN OFF TIME START AFTER RECIRCULATION OVER
   RUNG wire#powerrail
      Contact( "AlwaysTRUE" )
      { S7_Templates := "SrcType := Int" } EQ_Contact(in1 := "MODE SELECTION DB"."RO-2"."MODE BUFF", in2 := 1)
      { S7_Templates := "SrcType := Int" } EQ_Contact(in1 := "MODE SELECTION DB"."RO-2"."PROCESS BUFF", in2 := 2)
      { S7_Templates := "SrcType := Int" } EQ_Contact(in1 := "RO_2_LEVEL DB"."LEVEL HI RECIRC BUFF", in2 := 3)
      Contact( "TIMING_MIN_DB_10".DONE )
      Move(in := 4, out1 => "RO_2_LEVEL DB"."LEVEL HI RECIRC BUFF")
   END_RUNG
   // the same network as SCL:
   IF "AlwaysTRUE" AND ("MODE SELECTION DB"."RO-2"."MODE BUFF" = 1) AND ("MODE SELECTION DB"."RO-2"."PROCESS BUFF" = 2) AND ("RO_2_LEVEL DB"."LEVEL HI RECIRC BUFF" = 3) AND "TIMING_MIN_DB_10".DONE THEN
       "RO_2_LEVEL DB"."LEVEL HI RECIRC BUFF" := 4;
   END_IF;
END_REGION

REGION Network 18: AGAIN OFF TIME START AFTER RECIRCULATION OVER
   RUNG wire#powerrail
      Contact( "AlwaysTRUE" )
      { S7_Templates := "SrcType := Int" } EQ_Contact(in1 := "MODE SELECTION DB"."RO-2"."MODE BUFF", in2 := 1)
      { S7_Templates := "SrcType := Int" } EQ_Contact(in1 := "MODE SELECTION DB"."RO-2"."PROCESS BUFF", in2 := 2)
      { S7_Templates := "SrcType := Int" } EQ_Contact(in1 := "RO_2_LEVEL DB"."LEVEL HI RECIRC BUFF", in2 := 4)
      { S7_Templates := "time_type := Time" } "IEC_Timer_0_DB_95".TP(pt := T#2S, et =>)
      Move(in := 2, out1 => "RO_2_LEVEL DB"."LEVEL HI RECIRC BUFF")
   END_RUNG
   // the same network as SCL:
   "IEC_Timer_0_DB_95".TP(IN := "AlwaysTRUE" AND ("MODE SELECTION DB"."RO-2"."MODE BUFF" = 1) AND ("MODE SELECTION DB"."RO-2"."PROCESS BUFF" = 2) AND ("RO_2_LEVEL DB"."LEVEL HI RECIRC BUFF" = 4),
                          PT := T#2S);
   IF "IEC_Timer_0_DB_95".Q THEN "RO_2_LEVEL DB"."LEVEL HI RECIRC BUFF" := 2; END_IF;
END_REGION

REGION Network 19: REcirculation stop when level is normal
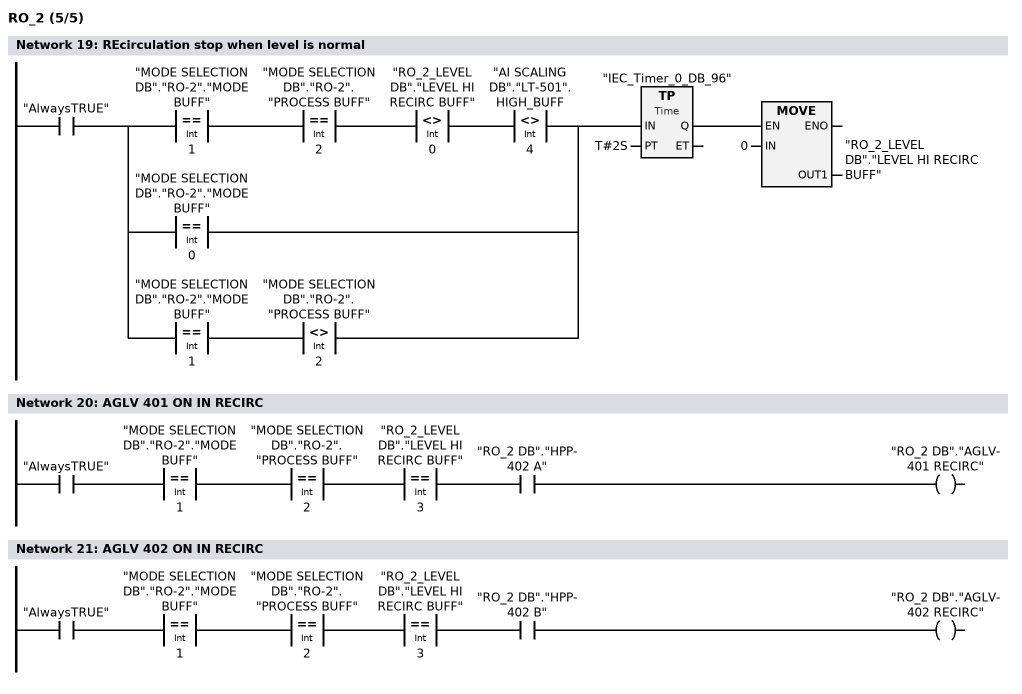
   RUNG wire#powerrail
      Contact( "AlwaysTRUE" )
      wire#w1
      { S7_Templates := "SrcType := Int" } EQ_Contact(in1 := "MODE SELECTION DB"."RO-2"."MODE BUFF", in2 := 1)
      { S7_Templates := "SrcType := Int" } EQ_Contact(in1 := "MODE SELECTION DB"."RO-2"."PROCESS BUFF", in2 := 2)
      { S7_Templates := "SrcType := Int" } NE_Contact(in1 := "RO_2_LEVEL DB"."LEVEL HI RECIRC BUFF", in2 := 0)
      { S7_Templates := "SrcType := Int" } NE_Contact(in1 := "AI SCALING DB"."LT-501".HIGH_BUFF, in2 := 4)
      wire#w2
      { S7_Templates := "time_type := Time" } "IEC_Timer_0_DB_96".TP(pt := T#2S, et =>)
      Move(in := 0, out1 => "RO_2_LEVEL DB"."LEVEL HI RECIRC BUFF")
   END_RUNG
   RUNG wire#w1
      { S7_Templates := "SrcType := Int" } EQ_Contact(in1 := "MODE SELECTION DB"."RO-2"."MODE BUFF", in2 := 0)
   END_RUNG wire#w2
   RUNG wire#w1
      { S7_Templates := "SrcType := Int" } EQ_Contact(in1 := "MODE SELECTION DB"."RO-2"."MODE BUFF", in2 := 1)
      { S7_Templates := "SrcType := Int" } NE_Contact(in1 := "MODE SELECTION DB"."RO-2"."PROCESS BUFF", in2 := 2)
   END_RUNG wire#w2
   // the same network as SCL:
   "IEC_Timer_0_DB_96".TP(IN := "AlwaysTRUE" AND ((("MODE SELECTION DB"."RO-2"."MODE BUFF" = 1) AND ("MODE SELECTION DB"."RO-2"."PROCESS BUFF" = 2) AND ("RO_2_LEVEL DB"."LEVEL HI RECIRC BUFF" <> 0) AND ("AI SCALING DB"."LT-501".HIGH_BUFF <> 4)) OR ("MODE SELECTION DB"."RO-2"."MODE BUFF" = 0) OR (("MODE SELECTION DB"."RO-2"."MODE BUFF" = 1) AND ("MODE SELECTION DB"."RO-2"."PROCESS BUFF" <> 2))),
                          PT := T#2S);
   IF "IEC_Timer_0_DB_96".Q THEN "RO_2_LEVEL DB"."LEVEL HI RECIRC BUFF" := 0; END_IF;
END_REGION

REGION Network 20: AGLV 401 ON IN RECIRC
   RUNG wire#powerrail
      Contact( "AlwaysTRUE" )
      { S7_Templates := "SrcType := Int" } EQ_Contact(in1 := "MODE SELECTION DB"."RO-2"."MODE BUFF", in2 := 1)
      { S7_Templates := "SrcType := Int" } EQ_Contact(in1 := "MODE SELECTION DB"."RO-2"."PROCESS BUFF", in2 := 2)
      { S7_Templates := "SrcType := Int" } EQ_Contact(in1 := "RO_2_LEVEL DB"."LEVEL HI RECIRC BUFF", in2 := 3)
      Contact( "RO_2 DB"."HPP-402 A" )
      Coil( "RO_2 DB"."AGLV-401 RECIRC" )
   END_RUNG
   // the same network as SCL:
   "RO_2 DB"."AGLV-401 RECIRC" := "AlwaysTRUE" AND ("MODE SELECTION DB"."RO-2"."MODE BUFF" = 1) AND ("MODE SELECTION DB"."RO-2"."PROCESS BUFF" = 2) AND ("RO_2_LEVEL DB"."LEVEL HI RECIRC BUFF" = 3) AND "RO_2 DB"."HPP-402 A";
END_REGION

REGION Network 21: AGLV 402 ON IN RECIRC
   RUNG wire#powerrail
      Contact( "AlwaysTRUE" )
      { S7_Templates := "SrcType := Int" } EQ_Contact(in1 := "MODE SELECTION DB"."RO-2"."MODE BUFF", in2 := 1)
      { S7_Templates := "SrcType := Int" } EQ_Contact(in1 := "MODE SELECTION DB"."RO-2"."PROCESS BUFF", in2 := 2)
      { S7_Templates := "SrcType := Int" } EQ_Contact(in1 := "RO_2_LEVEL DB"."LEVEL HI RECIRC BUFF", in2 := 3)
      Contact( "RO_2 DB"."HPP-402 B" )
      Coil( "RO_2 DB"."AGLV-402 RECIRC" )
   END_RUNG
   // the same network as SCL:
   "RO_2 DB"."AGLV-402 RECIRC" := "AlwaysTRUE" AND ("MODE SELECTION DB"."RO-2"."MODE BUFF" = 1) AND ("MODE SELECTION DB"."RO-2"."PROCESS BUFF" = 2) AND ("RO_2_LEVEL DB"."LEVEL HI RECIRC BUFF" = 3) AND "RO_2 DB"."HPP-402 B";
END_REGION
END_FUNCTION
